{attribute 'GeneratedUsingTerminal: ER8309-1022-0018'}
{attribute addProperty BoxType "ER8309-1022-0018"}
{attribute addProperty Id "Undervoltage_UsAT %I*BOOL1Undervoltage_UpAT %I*BOOL1"}
{attribute addProperty CRC "4226908324"}
{attribute addProperty Size "2"}
TYPE DEV_Inputs_FBF180A4 EXTENDS InputBase_8311D824 :
STRUCT
	{attribute addProperty Name "Undervoltage_Us"}
	Undervoltage_Us AT %I* : BOOL;
	{attribute addProperty Name "Undervoltage_Up"}
	Undervoltage_Up AT %I* : BOOL;
END_STRUCT
END_TYPE

(* stored: Version 1.2.0.0, ProductVersion 3.1.4024.9
   DUT DEV_Inputs_FBF180A4: Id {a0d17764-a6fe-468c-8fe5-d778498cfcd3} *)
